FUNCTION_BLOCK Test_TExecutionWhenBusy_SetAborted_RaisesEvent EXTENDS TUnitTestbase
VAR
    Execution : TExecution;
    Execution_EventHandler : TExecution_EventHandler;
END_VAR

// Setup...
Execution.FB_init(
    bInitRetains := FALSE,
    bInCopyCode  := FALSE);
Execution_EventHandler.FB_init(
    bInitRetains := FALSE,
    bInCopyCode  := FALSE);
    
// link handler to common execution events...
GlobalEvents.Event_OnAbort.ClearEventHandlers().AddEventHandler(Execution_EventHandler); 
GlobalEvents.Event_OnError.ClearEventHandlers().AddEventHandler(Execution_EventHandler);

// Test...
Execution.Start();
Execution.SetBusy();
Execution.SetAborted(); // raises error event

Assertion.AssertEquals_BOOL(
    Expected := TRUE,
    Actual   := Execution_EventHandler.AbortedEventRaised,
    VariableName  := 'EventHandler.AbortedEventRaised');
    
    
TestFinished();

END_FUNCTION_BLOCK

(* stored: Version 1.1.0.1, ProductVersion 3.1.4024.4
   POU Test_TExecutionWhenBusy_SetAborted_RaisesEvent: Id {e8be16a0-ec56-4944-b13e-7262c90d5c39}, SpecialFunc None *)
